FUNCTION_BLOCK GetTime
VAR_INPUT
	cycleTicks : REAL; // Unter SYSTEM -> TASKS eingestellte ticks
END_VAR
VAR_OUTPUT
	actTime : REAL;
END_VAR

VAR
	T : REAL;
	firstCall : BOOL := FALSE;
END_VAR

T  := ((cycleTicks*1.0) / 1000.0);
IF firstCall = FALSE THEN
	actTime := 0.0;
	firstCall := TRUE;
ELSE
	actTime := actTime + T;
END_IF

END_FUNCTION_BLOCK

(* stored: Version 1.1.0.1, ProductVersion 3.1.4022.10
   POU GetTime: Id {6b48b890-8388-4932-b767-5282b9a5d3f8}, SpecialFunc None *)
